FUNCTION F_MotorCalc : ST_MotorValues
VAR_INPUT
END_VAR
VAR
END_VAR


F_MotorCalc.bOverheat := TRUE;
F_MotorCalc.iEncoderPosition := 485;

END_FUNCTION

(* stored: Version 1.1.0.1, ProductVersion 3.1.4024.9
   POU F_MotorCalc: Id {7d943e7a-0a81-47f2-95ed-70a1a6eb75fd}, SpecialFunc None *)
